ABB RobotStudio station: Solution3.rsstn

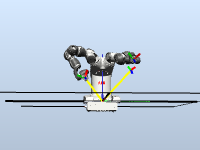
Station Solution3 (saved by RobotStudio format 3)
Controller IRB_14000_0.5kg_0.5m
  mechanical unit ROB_R: IRB14000_0.5_0.5_R, 6 joints, base frame (0, 0, 0) mm
  mechanical unit ROB_R_7: IRB14000_0.5_0.5_R, 1 joints, base frame (0, 0, 0) mm
  mechanical unit ROB_L: IRB14000_0.5_0.5_L, 6 joints, base frame (0, 0, 0) mm
  mechanical unit ROB_L_7: IRB14000_0.5_0.5_L, 1 joints, base frame (0, 0, 0) mm
Layout (positions relative to the parent item):
  - IRB14000_0.5_0.5_R [mechanism, from Robots\IRB14000_0.5_0.5_R.rslib] at (0, 0, 0) mm; joint values [1.1291, -0.7247, -1.7422, 0.4955, 2.3382, 1.0483, -0.9096] (rad or m)
  - IRB14000_0.5_0.5_L [mechanism, from Robots\IRB14000_0.5_0.5_L.rslib] at (0, 0, 0) mm; joint values [-2.2867, -0.9173, 0.603, -1.1108, 2.6121, 0.5731, 2.3647] (rad or m)
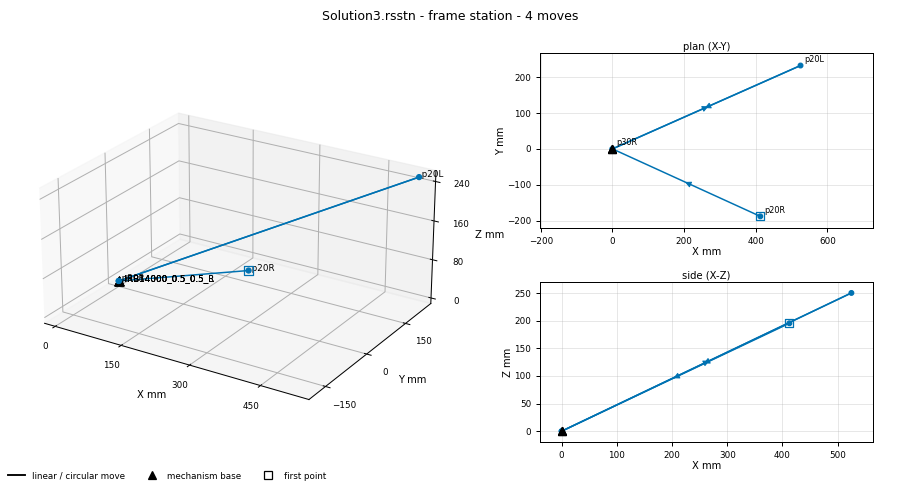
[picture p0: tool path of Solution3.rsstn in frame station, 4 of 4 moves have a stored position in this frame; points joined in program order, loops and branches not executed]
Targets, tools, work objects and paths stored in the station, written as RAPID:
! task T_ROB_R
MODULE MainModule
  VAR robtarget p20R:=[[412.53,-188.21,195.45],[0.0196523,0.791414,0.18309,0.582886],[0,1,-1,11],[150.954,9E9,9E9,9E9,9E9,9E9]];
  VAR robtarget p30R:=[[0,0,0],[1,0,0,0],[0,0,0,0],[9E9,9E9,9E9,9E9,9E9,9E9]];
  PROC main()
    ConfL \Off;
    MoveL p20R,v5000,z50,tool0;
    MoveL p30R,v5000,z50,tool0;
  ENDPROC
ENDMODULE

! task T_ROB_L
MODULE MainModule
  TASK PERS wobjdata Workobject_1:=[FALSE,TRUE,"",[[0,0,0],[1,0,0,0]],[[0,0,0],[1,0,0,0]]];
  PERS robtarget p20L:=[[524.76,232.69,250.37],[0.167465,0.793859,0.389036,0.436342],[-1,1,0,11],[152.059,9E9,9E9,9E9,9E9,9E9]];
  VAR robtarget p30L:=[[0,0,0],[1,0,0,0],[0,0,0,0],[9E9,9E9,9E9,9E9,9E9,9E9]];
  PROC main()
    ConfL \Off;
    MoveL p20L,v5000,z50,tool0\WObj:=Workobject_1;
    MoveL p30L,v1000,z50,tool0\WObj:=Workobject_1;
  ENDPROC
ENDMODULE

